FUNCTION_BLOCK T_ModuleCollectionOneIsNotInAskedStateReturnsCorrectResponse EXTENDS T_UnitTestBase
VAR
  list : T_SubModuleCollection(10);
  newModule, newModule2 : T_SubModuleMock; 
  actual1, actual2 : BOOL;
END_VAR

// Arrange
list.AddModule(newModule);
list.AddModule(newModule2);

//Act
newModule._Currentstate := Tc3_PackML_V2.E_PMLState.ePMLState_Completing;
newModule2._Currentstate := Tc3_PackML_V2.E_PMLState.ePMLState_Clearing;

//Assert
actual1 := NOT list.IsInAskedState(Tc3_PackML_V2.E_PMLState.ePMLState_Completing);

assertion.AssertEquals_BOOL(TRUE, actual1, 'actual1 := NOT list.IsInAskedState(Tc3_PackML_V2.E_PMLState.ePMLState_Completing');
TestFinished();

END_FUNCTION_BLOCK

(* stored: Version 1.1.0.1, ProductVersion 3.1.4024.12
   POU T_ModuleCollectionOneIsNotInAskedStateReturnsCorrectResponse: Id {8cc68880-e557-4213-8827-55e98921a759}, SpecialFunc None *)
